// TwinCAT 3 PLC project MC
// ProgramVersion: 3.1.4024.0
// libraries:
//   Tc2_MC2, * (Beckhoff Automation GmbH)
//   Tc2_MC2_Drive, * (Beckhoff Automation GmbH)
//   Tc2_Standard, * (Beckhoff Automation GmbH)
//   Tc2_System, * (Beckhoff Automation GmbH)
//   Tc3_Module, * (Beckhoff Automation GmbH)
//   VisuSymbols,3.5.10.0,System
// project tree:
//   DUTs/ ST_MC_Cmd.TcDUT (not stored), ST_MC_Status.TcDUT
//   / Gestore di visualizzazione.TcVMO (not stored), GlobalTextList.TcGTLO, PlcTask.TcTTO
//   GVLs/ GVL_SA.TcGVL
//   POUs/ MAIN.TcPOU, Motion.TcPOU
//   VISUs/ Visualization.TcVIS
// real-time tasks:
//   TASK PlcTask: cycle T#10ms, priority 20, ADS port 350
//   TASK PlcTask1: cycle T#10ms, priority 21, ADS port 351
// motion (NC):
//   TASK NC-Task 1 SAF: cycle T#2ms, priority 4, ADS port 501
//   TASK NC-Task 1 SVB: cycle T#10ms, priority 8, ADS port 511
//   AXIS Asse 1 (id 1)
//     OtherSettings: AllowMotionCmdToSlave=true
//     encoder EncType=1
//       Inc: RefSoftSyncMask=#x0000ffff
//     drive DrvType=24
//       Analog: TorqueSetpointScale=10, ScaleFactorActTorque=0.1
//       TimeComp: TaskDelayCycles=1
//     controller CtrType=1
//       CtrPara: PriorControlFactor=1
//         Observer: BandWidth=20
// I/O:
//   DEVICE Dispositivo 1 (EtherCAT), AmsNetId 5.71.198.244.2.1
//     Terminale 1 (EK1200) [EK1200-5000 EtherCAT Power supply (2A E-Bus)]
//       Terminale 2 (EL1008) [EL1008 8Ch. Dig. Input 24V, 3ms]
//       Terminale 3 (EL2008) [EL2008 8Ch. Dig. Output 24V, 0.5A]
//       Terminale 4 (EL3064) [EL3064 4Ch. Ana. Input 0-10V]
//       Terminale 5 (EL4002) [EL4002 2Ch. Ana. Output 0-10V, 12bit]
//       Terminale 6 (EL7031) [EL7031 1Ch. Stepper motor output stage (24V, 1.5A)]
//       Terminale 7 (EL3202) [EL3202 2Ch. Ana. Input PT100 (RTD)]
//       Terminale 8 (EL4022) [EL4022 2Ch. Ana. Output 4-20mA, 12bit]
//       Terminale 9 (EL9011) [EL9011 End Terminal]
// variable links:
//   NC-Task 1 SAF/Axes/Asse 1 <-> Device 1 (EtherCAT)/Term 1 (EK1200)/Term 6 (EL7031)
//     Drive/Inputs/In/nState1 @bit 3 <-> STM Status/Status/Error
//     Drive/Inputs/In/nState1 @bit 5 <-> STM Status/Status/Moving negative
//     Drive/Inputs/In/nState1 @bit 4 <-> STM Status/Status/Moving positive
//     Drive/Inputs/In/nState1 @bit 1 <-> STM Status/Status/Ready
//     Drive/Inputs/In/nState1 <-> STM Status/Status/Ready to enable
//     Drive/Inputs/In/nState1 @bit 6 <-> STM Status/Status/Torque reduced
//     Drive/Inputs/In/nState1 @bit 2 <-> STM Status/Status/Warning
//     Drive/Inputs/In/nState2 @bit 3 <-> STM Status/Status/Digital input 1
//     Drive/Inputs/In/nState2 @bit 4 <-> STM Status/Status/Digital input 2
//     Drive/Inputs/In/nState2 @bit 5 <-> STM Status/Status/Sync error
//     Drive/Inputs/In/nState2 @bit 7 <-> STM Status/Status/TxPDO Toggle
//     Drive/Inputs/In/nState4 @bit 1 <-> WcState/InputToggle
//     Drive/Inputs/In/nState4 <-> WcState/WcState
//     Drive/Outputs/Out/nCtrl1 <-> STM Control/Control/Enable
//     Drive/Outputs/Out/nCtrl1 @bit 2 <-> STM Control/Control/Reduce torque
//     Drive/Outputs/Out/nCtrl1 @bit 1 <-> STM Control/Control/Reset
//     Drive/Outputs/Out/nDataOut2[0] <-> STM Velocity/Velocity
//     Enc/Inputs/In/nDataIn1[0] <-> ENC Status compact/Counter value
//     Enc/Inputs/In/nDataIn2[0] <-> ENC Status compact/Latch value
//     Enc/Inputs/In/nState1 @bit 4 <-> ENC Status compact/Status/Counter overflow
//     Enc/Inputs/In/nState1 @bit 3 <-> ENC Status compact/Status/Counter underflow
//     Enc/Inputs/In/nState1 @bit 1 <-> ENC Status compact/Status/Latch extern valid
//     Enc/Inputs/In/nState1 @bit 2 <-> ENC Status compact/Status/Set counter done
//     Enc/Inputs/In/nState2 @bit 4 <-> ENC Status compact/Status/Status of extern latch
//     Enc/Inputs/In/nState2 @bit 5 <-> ENC Status compact/Status/Sync error
//     Enc/Inputs/In/nState2 @bit 7 <-> ENC Status compact/Status/TxPDO Toggle
//     Enc/Inputs/In/nState4 @bit 1 <-> WcState/InputToggle
//     Enc/Inputs/In/nState4 <-> WcState/WcState
//     Enc/Outputs/Out/nCtrl1 @bit 3 <-> ENC Control compact/Control/Enable latch extern on negative edge
//     Enc/Outputs/Out/nCtrl1 @bit 1 <-> ENC Control compact/Control/Enable latch extern on positive edge
//     Enc/Outputs/Out/nCtrl1 @bit 2 <-> ENC Control compact/Control/Set counter
//     Enc/Outputs/Out/nDataOut1[0] <-> ENC Control compact/Set counter value
//   MC/MC Instance <-> Device 1 (EtherCAT)/Term 1 (EK1200)/Term 2 (EL1008)
//     PlcTask Inputs/GVL_SA.bDigital_Inputs[{1..8}] <-> Channel {1..8}/Input  (8 links)
//   MC/MC Instance <-> Device 1 (EtherCAT)/Term 1 (EK1200)/Term 3 (EL2008)
//     PlcTask Outputs/GVL_SA.bDigital_Outputs[{1..8}] <-> Channel {1..8}/Output  (8 links)
//   MC/MC Instance <-> Device 1 (EtherCAT)/Term 1 (EK1200)/Term 5 (EL4002)
//     PlcTask Outputs/GVL_SA.bAnalog_Outputs[1] <-> AO Outputs Channel 1/Analog output
//     PlcTask Outputs/GVL_SA.bAnalog_Outputs[2] <-> AO Outputs Channel 2/Analog output
//   MC/MC Instance <-> NC-Task 1 SAF/Axes/Asse 1
//     PlcTask Inputs/GVL_SA.singleAxis.NcToPlc <-> Outputs/ToPlc
//     PlcTask Outputs/GVL_SA.singleAxis.PlcToNc <-> Inputs/FromPlc

CONFIGURATION MC
    RESOURCE PLC ON TwinCAT3
        TASK PlcTask(INTERVAL := T#10ms, PRIORITY := 21);
        PROGRAM MAIN WITH PlcTask : MAIN;
    END_RESOURCE
END_CONFIGURATION

// ---- DUTs/ST_MC_Status.TcDUT
TYPE ST_MC_Status :
STRUCT
	Status		: BOOL;
	Done		: BOOL;
	Busy		: BOOL;
	Error		: BOOL;
	Active		: BOOL;
	CadAborted	: BOOL;
	InVelocity	: BOOL;
	ErrorID		: UDINT;
END_STRUCT
END_TYPE

// ---- GVLs/GVL_SA.TcGVL
{attribute 'qualified_only'}
VAR_GLOBAL
	bDigital_Inputs AT %I* : ARRAY[1..8] OF BOOL;
	bDigital_Outputs AT %Q* : ARRAY[1..8] OF BOOL;
	
	bAnalog_Outputs AT %Q* : ARRAY[1..2] OF INT;
	Analog_Outputs_Values : ARRAY[1..2] OF REAL;
	
	// Single Axis 'SA'
	singleAxis : AXIS_REF;
	
	// Motion Control Function Block instance variable 'fbSA'
	fbSA_Reset				: MC_RESET;
	fbSA_Power				: MC_POWER;
	fbSA_Home				: MC_HOME;
	fbSA_Jog				: MC_JOG;
	fbSA_MoveVel1			: MC_MoveVelocity;
	fbSA_MoveVel2			: MC_MoveVelocity;
	fbSA_MoveRel1			: MC_MoveRelative;
	fbSA_MoveRel2			: MC_MoveRelative;
	fbSA_MoveAbs1			: MC_MoveAbsolute;
	fbSA_MoveAbs2			: MC_MoveAbsolute;
	fbSA_Stop				: MC_Stop;
	fbSA_Halt				: MC_Halt;
	
	fbSA_ReadStatus			: MC_ReadStatus;
	
	bSA_ResetExe			: BOOL;
	bSA_PowerEnCmd			: BOOL := TRUE;
	bSA_PowerEnPositive		: BOOL := TRUE;
	bSA_PowerEnNegative		: BOOL := TRUE;
	
	bSA_HomeExe				: BOOL;
	bSA_HomeCamInput		: BOOL;
	
	bSA_JogFwd				: BOOL;
	bSA_JogRev				: BOOL;
	
	bSA_Halt_Exe			: BOOL;
	bSA_Stop_Exe			: BOOL;
	
	stSA_VelCmd1			: ST_MC_Cmd;
	stSA_VelCmd2			: ST_MC_Cmd;
	stSA_RelCmd1			: ST_MC_Cmd;
	stSA_RelCmd2			: ST_MC_Cmd;
	stSA_AbsCmd1			: ST_MC_Cmd;
	stSA_AbsCmd2			: ST_MC_Cmd;
	
	lrSA_PowerOverride		: LREAL := 100;
	lrSA_HomePosition		: LREAL;
	lrSA_SetPosition		: LREAL;
	lrSA_JogVelocity		: LREAL;
	
	stSA_Reset				: ST_MC_Status;
	stSA_Power				: ST_MC_Status;
	stSA_Home				: ST_MC_Status;
	stSA_SetPosition		: ST_MC_Status;
	stSA_Jog				: ST_MC_Status;
	
	stSA_VelSts1			: ST_MC_Status;
	stSA_VelSts2			: ST_MC_Status;
	stSA_RelSts1			: ST_MC_Status;
	stSA_RelSts2			: ST_MC_Status;
	stSA_AbsSts1			: ST_MC_Status;
	stSA_AbsSts2			: ST_MC_Status;
	
	stSA_Halt				: ST_MC_Status;
	stSA_Stop				: ST_MC_Status;
END_VAR

// ---- POUs/MAIN.TcPOU
PROGRAM MAIN
VAR
END_VAR

Motion();

END_PROGRAM

// ---- POUs/Motion.TcPOU
PROGRAM Motion
VAR
	Timer1: TON;
	TImer2: TON;
	temp: REAL;
END_VAR

Motion.ReadStatus();
Motion.Velocity();
Motion.StartStop();
Motion.SingleAxis_LD();
Motion.MotionStatus();
Motion.Blink();
Motion.WriteAnalogValue();

ACTION Blink:
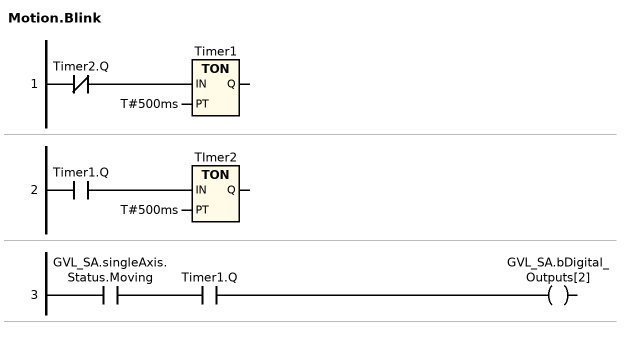
// NETWORK 1
Timer1(IN := NOT Timer2.Q, PT := T#500ms); // TON

// NETWORK 2
TImer2(IN := Timer1.Q, PT := T#500ms); // TON

// NETWORK 3
GVL_SA.bDigital_Outputs[2] := GVL_SA.singleAxis.Status.Moving AND Timer1.Q;
END_ACTION

ACTION MotionStatus:
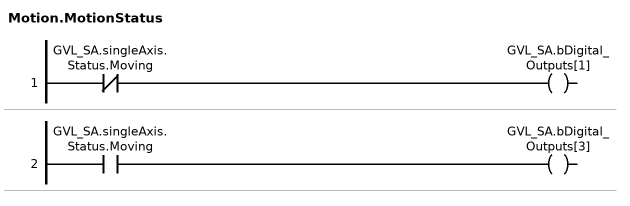
// NETWORK 1
GVL_SA.bDigital_Outputs[1] := NOT GVL_SA.singleAxis.Status.Moving;

// NETWORK 2
GVL_SA.bDigital_Outputs[3] := GVL_SA.singleAxis.Status.Moving;
END_ACTION

ACTION ReadStatus:
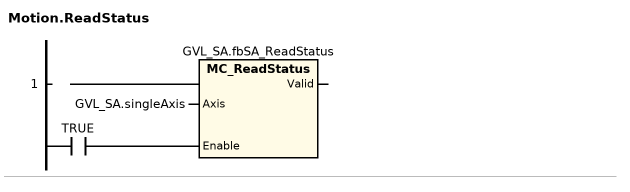
// NETWORK 1
GVL_SA.fbSA_ReadStatus(Axis := GVL_SA.singleAxis, Enable := TRUE); // MC_ReadStatus
END_ACTION

METHOD SingleAxis_LD : BOOL
VAR_INPUT
END_VAR
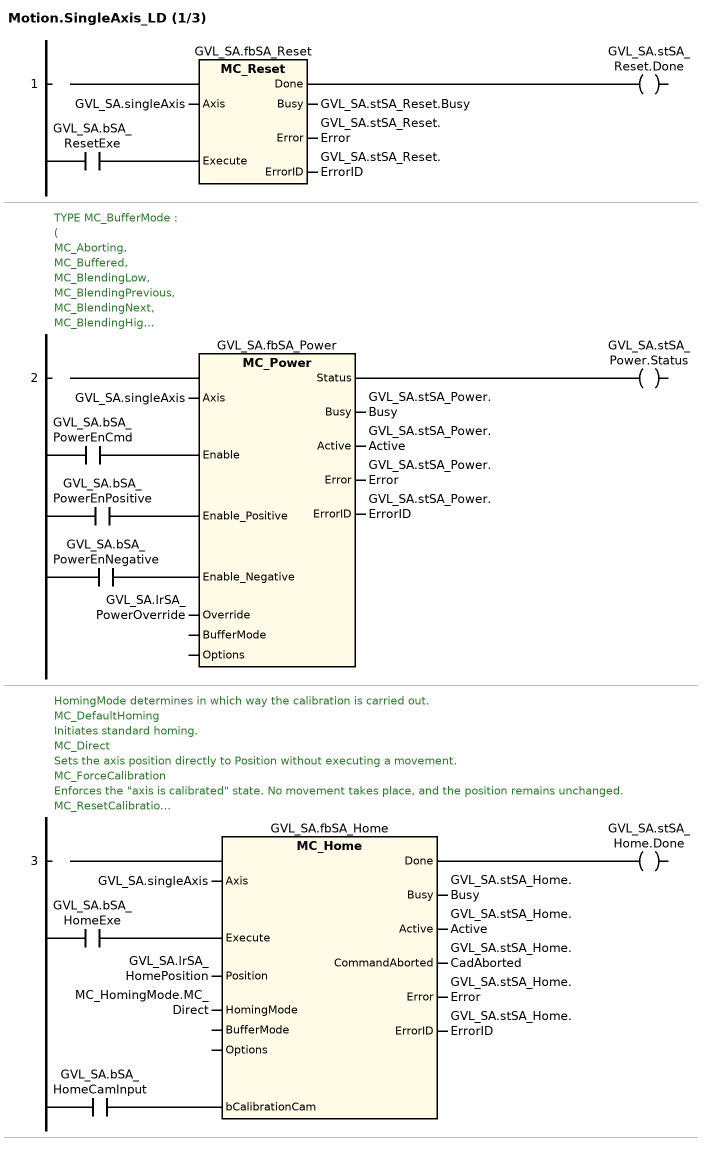
// NETWORK 1
GVL_SA.fbSA_Reset(
    Axis := GVL_SA.singleAxis,
    Execute := GVL_SA.bSA_ResetExe,
    Busy => GVL_SA.stSA_Reset.Busy,
    Error => GVL_SA.stSA_Reset.Error,
    ErrorID => GVL_SA.stSA_Reset.ErrorID); // MC_Reset
GVL_SA.stSA_Reset.Done := GVL_SA.fbSA_Reset.Done;

// NETWORK 2
// TYPE MC_BufferMode :
// (
//     MC_Aborting,
//     MC_Buffered,
//     MC_BlendingLow,
//     MC_BlendingPrevious,
//     MC_BlendingNext,
//     MC_BlendingHigh
// );
// END_TYPE
GVL_SA.fbSA_Power(
    Axis := GVL_SA.singleAxis,
    Enable := GVL_SA.bSA_PowerEnCmd,
    Enable_Positive := GVL_SA.bSA_PowerEnPositive,
    Enable_Negative := GVL_SA.bSA_PowerEnNegative,
    Override := GVL_SA.lrSA_PowerOverride,
    Busy => GVL_SA.stSA_Power.Busy,
    Active => GVL_SA.stSA_Power.Active,
    Error => GVL_SA.stSA_Power.Error,
    ErrorID => GVL_SA.stSA_Power.ErrorID); // MC_Power
GVL_SA.stSA_Power.Status := GVL_SA.fbSA_Power.Status;

// NETWORK 3
// HomingMode determines in which way the calibration is carried out.
//
// MC_DefaultHoming
// Initiates standard homing.
// MC_Direct
// Sets the axis position directly to Position without executing a movement.
// MC_ForceCalibration
// Enforces the "axis is calibrated" state. No movement takes place, and the position remains unchanged.
// MC_ResetCalibration
// Resets the calibration state of the axis. No movement takes place, and the position remains unchanged.
GVL_SA.fbSA_Home(
    Axis := GVL_SA.singleAxis,
    Execute := GVL_SA.bSA_HomeExe,
    Position := GVL_SA.lrSA_HomePosition,
    HomingMode := MC_HomingMode.MC_Direct,
    bCalibrationCam := GVL_SA.bSA_HomeCamInput,
    Busy => GVL_SA.stSA_Home.Busy,
    Active => GVL_SA.stSA_Home.Active,
    CommandAborted => GVL_SA.stSA_Home.CadAborted,
    Error => GVL_SA.stSA_Home.Error,
    ErrorID => GVL_SA.stSA_Home.ErrorID); // MC_Home
GVL_SA.stSA_Home.Done := GVL_SA.fbSA_Home.Done;

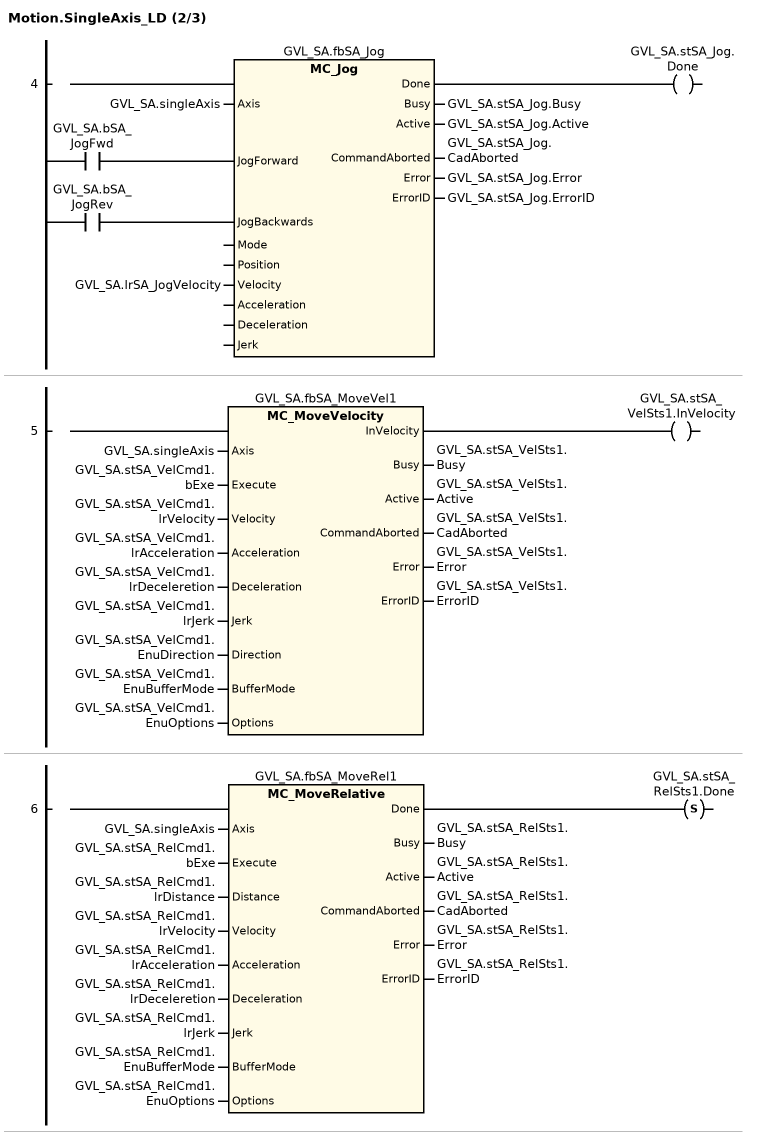
// NETWORK 4
GVL_SA.fbSA_Jog(
    Axis := GVL_SA.singleAxis,
    JogForward := GVL_SA.bSA_JogFwd,
    JogBackwards := GVL_SA.bSA_JogRev,
    Velocity := GVL_SA.lrSA_JogVelocity,
    Busy => GVL_SA.stSA_Jog.Busy,
    Active => GVL_SA.stSA_Jog.Active,
    CommandAborted => GVL_SA.stSA_Jog.CadAborted,
    Error => GVL_SA.stSA_Jog.Error,
    ErrorID => GVL_SA.stSA_Jog.ErrorID); // MC_Jog
GVL_SA.stSA_Jog.Done := GVL_SA.fbSA_Jog.Done;

// NETWORK 5
GVL_SA.fbSA_MoveVel1(
    Axis := GVL_SA.singleAxis,
    Execute := GVL_SA.stSA_VelCmd1.bExe,
    Velocity := GVL_SA.stSA_VelCmd1.lrVelocity,
    Acceleration := GVL_SA.stSA_VelCmd1.lrAcceleration,
    Deceleration := GVL_SA.stSA_VelCmd1.lrDeceleretion,
    Jerk := GVL_SA.stSA_VelCmd1.lrJerk,
    Direction := GVL_SA.stSA_VelCmd1.EnuDirection,
    BufferMode := GVL_SA.stSA_VelCmd1.EnuBufferMode,
    Options := GVL_SA.stSA_VelCmd1.EnuOptions,
    Busy => GVL_SA.stSA_VelSts1.Busy,
    Active => GVL_SA.stSA_VelSts1.Active,
    CommandAborted => GVL_SA.stSA_VelSts1.CadAborted,
    Error => GVL_SA.stSA_VelSts1.Error,
    ErrorID => GVL_SA.stSA_VelSts1.ErrorID); // MC_MoveVelocity
GVL_SA.stSA_VelSts1.InVelocity := GVL_SA.fbSA_MoveVel1.InVelocity;

// NETWORK 6
GVL_SA.fbSA_MoveRel1(
    Axis := GVL_SA.singleAxis,
    Execute := GVL_SA.stSA_RelCmd1.bExe,
    Distance := GVL_SA.stSA_RelCmd1.lrDistance,
    Velocity := GVL_SA.stSA_RelCmd1.lrVelocity,
    Acceleration := GVL_SA.stSA_RelCmd1.lrAcceleration,
    Deceleration := GVL_SA.stSA_RelCmd1.lrDeceleretion,
    Jerk := GVL_SA.stSA_RelCmd1.lrJerk,
    BufferMode := GVL_SA.stSA_RelCmd1.EnuBufferMode,
    Options := GVL_SA.stSA_RelCmd1.EnuOptions,
    Busy => GVL_SA.stSA_RelSts1.Busy,
    Active => GVL_SA.stSA_RelSts1.Active,
    CommandAborted => GVL_SA.stSA_RelSts1.CadAborted,
    Error => GVL_SA.stSA_RelSts1.Error,
    ErrorID => GVL_SA.stSA_RelSts1.ErrorID); // MC_MoveRelative
GVL_SA.stSA_RelSts1.Done S= GVL_SA.fbSA_MoveRel1.Done;

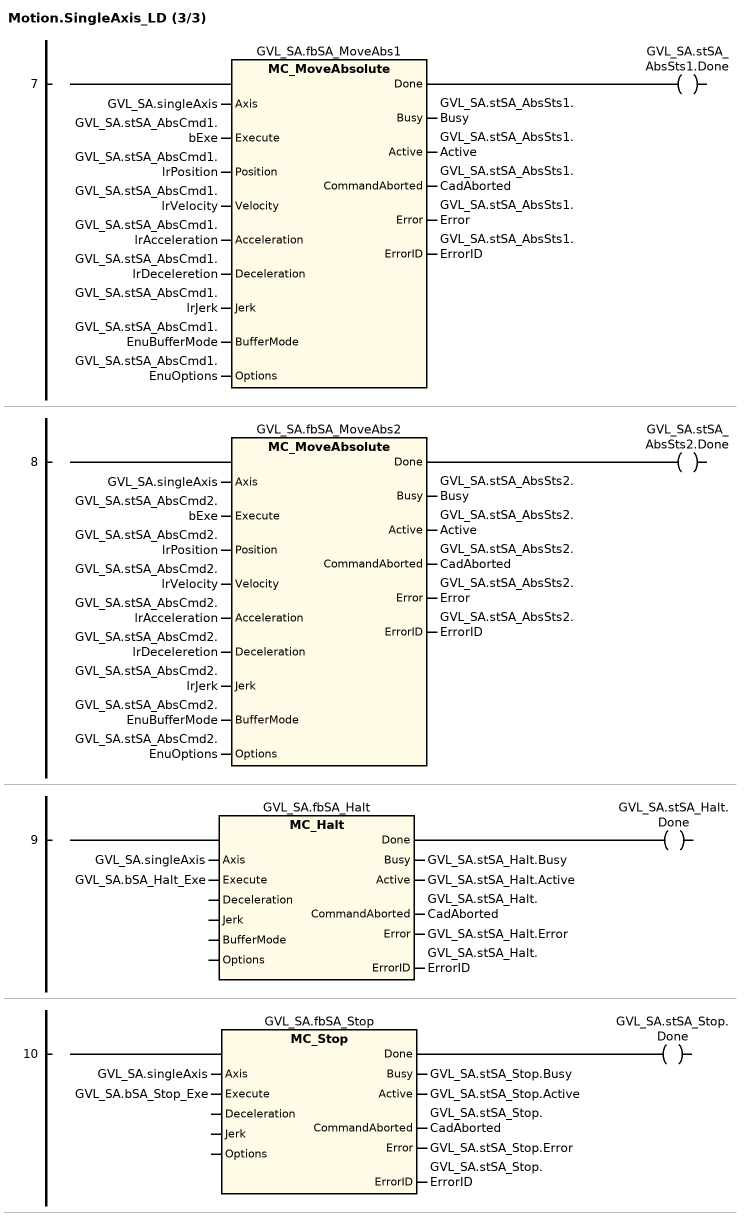
// NETWORK 7
GVL_SA.fbSA_MoveAbs1(
    Axis := GVL_SA.singleAxis,
    Execute := GVL_SA.stSA_AbsCmd1.bExe,
    Position := GVL_SA.stSA_AbsCmd1.lrPosition,
    Velocity := GVL_SA.stSA_AbsCmd1.lrVelocity,
    Acceleration := GVL_SA.stSA_AbsCmd1.lrAcceleration,
    Deceleration := GVL_SA.stSA_AbsCmd1.lrDeceleretion,
    Jerk := GVL_SA.stSA_AbsCmd1.lrJerk,
    BufferMode := GVL_SA.stSA_AbsCmd1.EnuBufferMode,
    Options := GVL_SA.stSA_AbsCmd1.EnuOptions,
    Busy => GVL_SA.stSA_AbsSts1.Busy,
    Active => GVL_SA.stSA_AbsSts1.Active,
    CommandAborted => GVL_SA.stSA_AbsSts1.CadAborted,
    Error => GVL_SA.stSA_AbsSts1.Error,
    ErrorID => GVL_SA.stSA_AbsSts1.ErrorID); // MC_MoveAbsolute
GVL_SA.stSA_AbsSts1.Done := GVL_SA.fbSA_MoveAbs1.Done;

// NETWORK 8
GVL_SA.fbSA_MoveAbs2(
    Axis := GVL_SA.singleAxis,
    Execute := GVL_SA.stSA_AbsCmd2.bExe,
    Position := GVL_SA.stSA_AbsCmd2.lrPosition,
    Velocity := GVL_SA.stSA_AbsCmd2.lrVelocity,
    Acceleration := GVL_SA.stSA_AbsCmd2.lrAcceleration,
    Deceleration := GVL_SA.stSA_AbsCmd2.lrDeceleretion,
    Jerk := GVL_SA.stSA_AbsCmd2.lrJerk,
    BufferMode := GVL_SA.stSA_AbsCmd2.EnuBufferMode,
    Options := GVL_SA.stSA_AbsCmd2.EnuOptions,
    Busy => GVL_SA.stSA_AbsSts2.Busy,
    Active => GVL_SA.stSA_AbsSts2.Active,
    CommandAborted => GVL_SA.stSA_AbsSts2.CadAborted,
    Error => GVL_SA.stSA_AbsSts2.Error,
    ErrorID => GVL_SA.stSA_AbsSts2.ErrorID); // MC_MoveAbsolute
GVL_SA.stSA_AbsSts2.Done := GVL_SA.fbSA_MoveAbs2.Done;

// NETWORK 9
GVL_SA.fbSA_Halt(
    Axis := GVL_SA.singleAxis,
    Execute := GVL_SA.bSA_Halt_Exe,
    Busy => GVL_SA.stSA_Halt.Busy,
    Active => GVL_SA.stSA_Halt.Active,
    CommandAborted => GVL_SA.stSA_Halt.CadAborted,
    Error => GVL_SA.stSA_Halt.Error,
    ErrorID => GVL_SA.stSA_Halt.ErrorID); // MC_Halt
GVL_SA.stSA_Halt.Done := GVL_SA.fbSA_Halt.Done;

// NETWORK 10
GVL_SA.fbSA_Stop(
    Axis := GVL_SA.singleAxis,
    Execute := GVL_SA.bSA_Stop_Exe,
    Busy => GVL_SA.stSA_Stop.Busy,
    Active => GVL_SA.stSA_Stop.Active,
    CommandAborted => GVL_SA.stSA_Stop.CadAborted,
    Error => GVL_SA.stSA_Stop.Error,
    ErrorID => GVL_SA.stSA_Stop.ErrorID); // MC_Stop
GVL_SA.stSA_Stop.Done := GVL_SA.fbSA_Stop.Done;
END_METHOD

METHOD StartStop : BOOL
VAR_INPUT
END_VAR
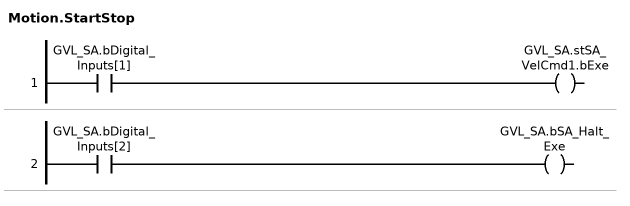
// NETWORK 1
GVL_SA.stSA_VelCmd1.bExe := GVL_SA.bDigital_Inputs[1];

// NETWORK 2
GVL_SA.bSA_Halt_Exe := GVL_SA.bDigital_Inputs[2];
END_METHOD

ACTION Velocity:
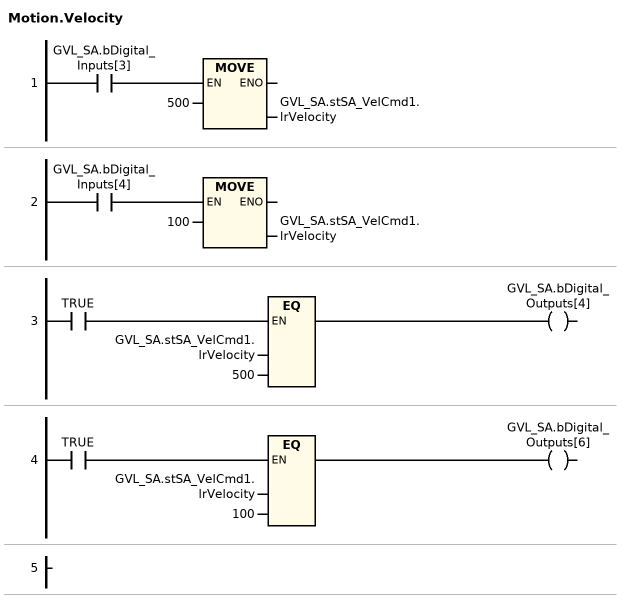
// NETWORK 1
IF GVL_SA.bDigital_Inputs[3] THEN GVL_SA.stSA_VelCmd1.lrVelocity := 500; END_IF

// NETWORK 2
IF GVL_SA.bDigital_Inputs[4] THEN GVL_SA.stSA_VelCmd1.lrVelocity := 100; END_IF

// NETWORK 3
GVL_SA.bDigital_Outputs[4] := GVL_SA.stSA_VelCmd1.lrVelocity = 500;

// NETWORK 4
GVL_SA.bDigital_Outputs[6] := GVL_SA.stSA_VelCmd1.lrVelocity = 100;

// NETWORK 5
END_ACTION

ACTION WriteAnalogValue:
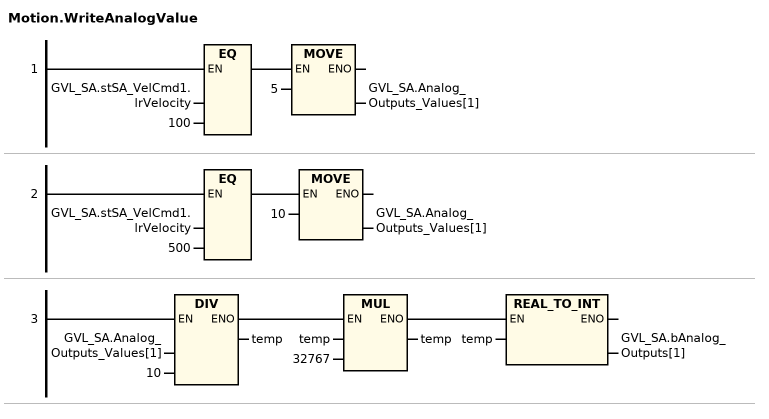
// NETWORK 1
IF GVL_SA.stSA_VelCmd1.lrVelocity = 100 THEN GVL_SA.Analog_Outputs_Values[1] := 5; END_IF

// NETWORK 2
IF GVL_SA.stSA_VelCmd1.lrVelocity = 500 THEN GVL_SA.Analog_Outputs_Values[1] := 10; END_IF

// NETWORK 3
temp := GVL_SA.Analog_Outputs_Values[1] / 10;
temp := temp * 32767;
GVL_SA.bAnalog_Outputs[1] := REAL_TO_INT(temp);
END_ACTION

END_PROGRAM

// ---- GlobalTextList.TcGTLO
TEXTLIST GlobalTextList
  273 = '%d'
  746 = 'Motore in funzione'
  561 = 'Velocità'
  844 = 'Velocità attuale'
  462 = 'Velocità impostata'
END_TEXTLIST

// ---- VISUs/Visualization.TcVIS
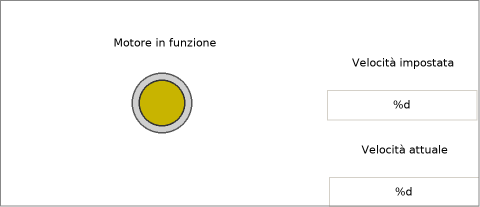
VISUALIZATION Visualization  // 480x207
    Lamp1 (127,68 70x70), variable: GVL_SA.singleAxis.Status.Moving, style: Lamp-Lamp1-Yellow
    Textfield (327,90 150x30), "%d", text variable: GVL_SA.stSA_VelCmd1.lrVelocity
    Label (328,48 150x30), "Velocità impostata"
    Label (90,28 150x30), "Motore in funzione"
    Textfield (329,177 150x30), "%d", text variable: GVL_SA.singleAxis.NcToPlc.ActVelo
    Label (330,135 150x30), "Velocità attuale"
END_VISUALIZATION
